Yaskawa INFORM job: slope_planes_program_2.JBI

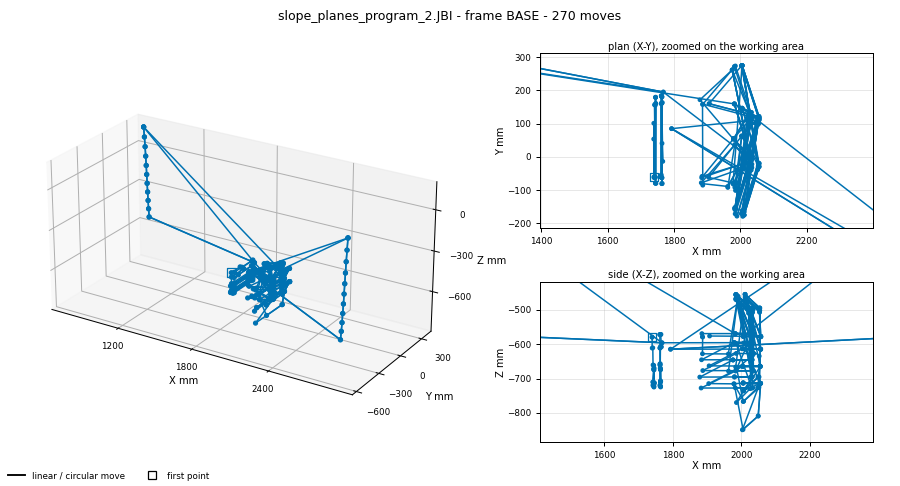
[picture p0: tool path of slope_planes_program_2.JBI in frame BASE, 270 of 278 moves have a stored position in this frame; points joined in program order, loops and branches not executed]
/JOB
//NAME slope_planes_program_2
//POS
///NPOS 270,0,270,0,0,0
///TOOL 0
///POSTYPE BASE
///RECTAN
///RCONF 0,0,0,0,0,0,0,0,0,0,0,0,0,0,0,0,0,0,0,0,0,0,0,0
C00000=1739.260769,-60.871235,-578.989580,5.000000,-89.172678,-175.000000
C00001=1739.028106,53.830840,-579.601277,5.000000,-89.172678,-175.000000
C00002=1739.284791,101.372352,-611.275362,5.000000,-89.172678,-175.000000
C00003=1741.092847,-62.556544,-610.379835,5.000000,-89.172678,-175.000000
C00004=1741.778439,-62.282291,-660.377305,5.000000,-89.172678,-175.000000
C00005=1743.760127,155.636241,-661.504448,5.000000,-89.172678,-175.000000
C00006=1744.673230,178.979946,-711.620985,5.000000,-89.172678,-175.000000
C00007=1740.845557,-59.386621,-710.412050,5.000000,-89.172678,-175.000000
C00008=1743.319095,-61.226324,-673.769949,180.000000,-60.000000,0.000000
C00009=1744.726413,180.007491,-675.029042,180.000000,-60.000000,0.000000
C00010=1744.389872,179.342411,-725.036290,180.000000,-60.000000,0.000000
C00011=1744.215946,-60.947521,-723.764393,180.000000,-60.000000,0.000000
C00012=1884.339610,-58.334513,-568.930098,5.000000,-89.675586,-175.000000
C00013=2032.194970,-12.730020,-568.874909,5.000000,-89.934306,115.240173
C00014=1985.150049,-157.658308,-456.347117,175.000000,-47.917446,5.000000
C00015=2029.012249,-22.244464,-494.713723,175.000000,-65.510944,-60.519673
C00016=2032.887715,-5.143099,-568.885585,5.000000,-89.935736,114.990048
C00017=1981.779671,159.548677,-569.132654,140.189389,-89.999999,5.000000
C00018=2032.201723,-8.373668,-568.883888,-5.000000,-89.934178,115.262595
C00019=1985.641519,-153.780863,-671.511595,-5.000000,-47.740214,-174.961836
C00020=2031.527886,117.688240,-633.513782,5.000000,-65.336014,119.271243
C00021=2033.332423,134.046107,-569.170815,5.000000,-89.932211,115.609393
C00022=1981.779671,159.548677,-569.132654,140.189389,-89.999999,5.000000
C00023=2032.199883,-9.878738,-568.880782,-5.000000,-89.934223,115.254638
C00024=1985.190754,-154.787790,-456.233996,175.000000,-47.916014,5.000000
C00025=2029.085818,-16.497927,-494.609987,175.000000,-65.511330,-60.517922
C00026=2032.946568,0.595729,-568.897051,-5.000000,-89.935689,114.998332
C00027=1981.779671,159.548677,-569.132654,140.189389,-89.999999,5.000000
C00028=2032.202884,-7.055256,-568.886612,5.000000,-89.934137,115.269757
C00029=1985.295997,-151.982336,-466.966556,175.000000,-47.913519,5.000000
C00030=2030.706860,98.840001,-505.585974,175.000000,-65.518281,-60.512478
C00031=2033.557205,115.500512,-569.130752,5.000000,-89.933364,115.405725
C00032=1981.779671,159.548677,-569.132654,140.189389,-89.999999,5.000000
C00033=747.892171,350.982236,154.177497,-16.058325,-5.000000,-175.000000
C00034=747.959774,350.940433,154.234940,-16.059565,-5.000000,-175.000000
C00035=745.781823,361.597631,74.788692,-16.556562,-5.272278,-175.000000
C00036=744.195610,370.293866,-2.453873,-17.385711,-8.680619,-175.000000
C00037=742.808280,377.250152,-77.638846,-18.568266,-11.941707,-175.000000
C00038=742.161890,382.679607,-150.970735,-20.134608,-15.003112,-174.578249
C00039=742.158513,386.664759,-222.101724,-22.108789,-17.810032,-172.917166
C00040=742.703577,389.417825,-291.287358,-24.515478,-20.302282,-171.008190
C00041=744.341698,390.973681,-358.590204,-27.364597,-22.407407,-168.839370
C00042=746.902560,391.345145,-424.326844,-30.640421,-24.064136,-166.421059
C00043=750.369947,390.762543,-488.235309,-34.306804,-25.187057,-163.807677
C00044=755.166090,389.038049,-550.708088,-5.000000,-44.999700,137.718258
C00045=1767.915992,195.255561,-595.676951,140.189389,-89.999999,5.000000
C00046=747.892171,350.982236,154.177497,-16.058325,-5.000000,-175.000000
C00047=747.959774,350.940433,154.234940,-16.059565,-5.000000,-175.000000
C00048=745.781823,361.597631,74.788692,-16.556562,-5.272278,-175.000000
C00049=744.195610,370.293866,-2.453873,-17.385711,-8.680619,-175.000000
C00050=742.808280,377.250152,-77.638846,-18.568266,-11.941707,-175.000000
C00051=742.161890,382.679607,-150.970735,-20.134608,-15.003112,-174.578249
C00052=742.158513,386.664759,-222.101724,-22.108789,-17.810032,-172.917166
C00053=742.703577,389.417825,-291.287358,-24.515478,-20.302282,-171.008190
C00054=744.341698,390.973681,-358.590204,-27.364597,-22.407407,-168.839370
C00055=746.902560,391.345145,-424.326844,-30.640421,-24.064136,-166.421059
C00056=750.369947,390.762543,-488.235309,-34.306804,-25.187057,-163.807677
C00057=755.166090,389.038049,-550.708088,-5.000000,-44.999700,137.718258
C00058=1767.915992,195.255561,-595.676951,140.189389,-89.999999,5.000000
C00059=2030.623854,-5.286374,-595.315431,-5.000000,-89.935275,115.070495
C00060=2026.211755,-22.498761,-494.867644,175.000000,-65.570252,-60.256248
C00061=1983.548198,-157.719294,-455.776356,-175.000000,-47.616753,5.000000
C00062=2030.498190,-12.647404,-595.301228,5.000000,-89.935007,115.117369
C00063=1978.860133,54.290550,-595.350371,140.189389,-89.999999,5.000000
C00064=2030.811257,134.553300,-595.601250,5.000000,-89.935056,115.108749
C00065=2026.562431,117.353936,-508.906406,175.000000,-65.570991,-60.254135
C00066=1983.639451,-153.364957,-469.532259,175.000000,-47.614280,5.000000
C00067=2030.498822,-8.269798,-595.310214,-5.000000,-89.934987,115.120777
C00068=1978.860133,54.290550,-595.350371,140.189389,-89.999999,5.000000
C00069=2030.633524,0.460796,-595.327163,5.000000,-89.935271,115.071236
C00070=2026.217270,-16.752716,-494.764546,-175.000000,-65.570746,-60.254012
C00071=1983.558465,-154.850766,-455.660837,-175.000000,-47.613977,5.000000
C00072=2030.498681,-9.782412,-595.307109,-5.000000,-89.934994,115.119567
C00073=1978.860133,54.290550,-595.350371,140.189389,-89.999999,5.000000
C00074=2030.796749,115.788780,-595.562819,5.000000,-89.935111,115.099123
C00075=2026.507696,98.585677,-505.732438,-175.000000,-65.571101,-60.254277
C00076=1983.625135,-152.033444,-466.398636,175.000000,-47.614083,5.000000
C00077=2030.498875,-6.944594,-595.312935,-5.000000,-89.934981,115.121867
C00078=1978.860133,54.290550,-595.350371,140.189389,-89.999999,5.000000
C00079=1883.381965,-62.373142,-645.345158,5.000000,-89.675586,-175.000000
C00080=2030.706335,-12.453119,-645.300320,5.000000,-89.936548,114.848944
C00081=1983.892004,-157.801574,-454.648135,175.000000,-47.028479,5.000000
C00082=2024.235575,-22.997670,-495.135127,175.000000,-65.680346,-59.751352
C00083=2029.274030,-5.746385,-645.324257,-5.000000,-89.933449,115.390836
C00084=1975.194699,261.761272,-645.797441,140.189389,-89.999999,5.000000
C00085=2030.702768,-8.032373,-645.309265,-5.000000,-89.936754,114.813150
C00086=1983.880333,-153.447358,-468.409969,175.000000,-47.028789,5.000000
C00087=2021.484525,116.857168,-509.189861,-175.000000,-65.680404,-59.751589
C00088=2027.006358,134.400777,-645.623562,5.000000,-89.934799,115.153719
C00089=1975.194699,261.761272,-645.797441,140.189389,-89.999999,5.000000
C00090=2030.703176,-9.560304,-645.306180,-5.000000,-89.936681,114.825864
C00091=1983.830510,-154.932885,-454.540310,175.000000,-47.029501,5.000000
C00092=2024.119139,-17.248911,-495.031310,175.000000,-65.680234,-59.751883
C00093=2029.170564,0.007674,-645.336620,5.000000,-89.933479,115.385431
C00094=1975.194699,261.761272,-645.797441,140.189389,-89.999999,5.000000
C00095=1878.225019,172.061174,-695.855961,5.000000,-89.675586,-175.000000
C00096=2029.216695,-5.923005,-695.325374,5.000000,-89.933075,115.456764
C00097=2023.915349,-23.060021,-495.167917,175.000000,-65.693651,-59.689227
C00098=1983.858125,-157.808143,-454.509625,175.000000,-46.955640,5.000000
C00099=2030.861995,-12.538689,-695.300110,-5.000000,-89.936636,114.833532
C00100=1979.614915,54.878233,-695.349115,140.189389,-89.999999,5.000000
C00101=2026.506483,134.201278,-695.627221,-5.000000,-89.934303,115.240728
C00102=2020.769283,116.793372,-509.225484,175.000000,-65.693966,-59.688064
C00103=1983.837631,-153.454231,-468.268165,175.000000,-46.954194,5.000000
C00104=2030.854062,-8.114311,-695.309074,5.000000,-89.936862,114.794410
C00105=1979.614915,54.878233,-695.349115,140.189389,-89.999999,5.000000
C00106=2029.096697,-0.169123,-695.337832,5.000000,-89.933104,115.451530
C00107=2025.415227,-17.647329,-729.697883,180.000000,-60.000000,0.000000
C00108=1985.252939,-155.837043,-770.197594,180.000000,-60.000000,0.000000
C00109=2030.855920,-9.643522,-695.305982,-5.000000,-89.936782,114.808298
C00110=1979.614915,54.878233,-695.349115,140.189389,-89.999999,5.000000
C00111=1745.307470,160.600706,-712.870295,175.000000,-89.223717,-5.000000
C00112=1745.747004,-79.714542,-714.068825,175.000000,-89.223717,-5.000000
C00113=1743.887926,-78.841577,-670.993376,180.000000,-60.000000,0.000000
C00114=1744.996879,160.942797,-669.818462,180.000000,-60.000000,0.000000
C00115=1741.316004,156.853693,-719.794086,180.000000,-60.000000,0.000000
C00116=1744.102037,-78.968875,-721.002114,180.000000,-60.000000,0.000000
C00117=1885.863395,158.182403,-578.045584,175.000000,-89.336646,-5.000000
C00118=1886.650424,-84.961125,-579.077831,175.000000,-89.336646,-5.000000
C00119=1886.044276,-80.394228,-627.842130,175.000000,-89.336646,-5.000000
C00120=1961.540570,-88.734620,-628.321589,-5.000000,-89.772434,-156.563433
C00121=1989.769528,-39.136527,-460.340640,175.000000,-47.501225,5.075310
C00122=2033.646978,102.591245,-498.881535,175.000000,-65.273893,-60.828128
C00123=2035.991453,119.891152,-627.326416,175.000000,-89.867726,-65.037930
C00124=1984.737237,273.797954,-626.863225,140.054684,-90.000000,5.000000
C00125=1887.028142,158.913088,-676.850323,175.000000,-89.336646,-5.000000
C00126=2034.825328,120.042378,-677.315653,175.000000,-89.867100,-64.984445
C00127=2032.776243,102.409388,-498.967851,175.000000,-65.312424,-60.640081
C00128=1989.800549,-39.182084,-459.925091,175.000000,-47.287692,5.116560
C00129=1962.013642,-91.664127,-678.436686,5.000000,-89.725460,-155.249492
C00130=1982.938067,36.726704,-677.843770,140.054684,-90.000000,5.000000
C00131=2034.622962,-22.049069,-677.911343,175.000000,-89.867279,-64.999786
C00132=2032.449640,-39.666207,-507.153666,-175.000000,-65.312498,-60.640202
C00133=1989.478498,-178.135948,-468.098074,175.000000,-47.287911,5.116557
C00134=2034.502364,-31.953303,-677.951280,175.000000,-89.866766,-64.955929
C00135=1982.938067,36.726704,-677.843770,140.054684,-90.000000,5.000000
C00136=1882.142247,-77.828377,-727.793743,175.000000,-89.336646,-5.000000
C00137=2030.206063,-25.652685,-727.877558,175.000000,-89.864872,-64.793536
C00138=1984.108354,-171.256741,-597.047291,175.000000,-47.594353,5.056180
C00139=2030.104031,98.022525,-634.851776,-175.000000,-65.256846,-60.910378
C00140=2032.751310,115.122397,-727.316773,-175.000000,-89.868050,-65.065618
C00141=1981.628604,272.117578,-726.841892,140.054684,-90.000000,5.000000
C00142=1906.927979,159.938160,-576.005760,175.000000,-88.730027,-5.000000
C00143=2055.823639,120.996000,-576.901902,-175.000000,-89.740938,-65.240948
C00144=2053.106317,103.764595,-494.268027,-175.000000,-65.230923,-61.019642
C00145=2010.474853,-34.355523,-454.220693,175.000000,-46.647438,5.000000
C00146=2056.406479,111.482410,-576.995998,175.000000,-89.745867,-65.461252
C00147=2005.209070,146.661390,-577.065002,139.450504,-90.000000,5.000000
C00148=2055.842019,116.746081,-576.937074,-175.000000,-89.740871,-65.237935
C00149=2052.989906,99.574050,-500.952961,175.000000,-65.230260,-61.021788
C00150=2011.168552,-174.704832,-462.043828,175.000000,-46.649165,5.000000
C00151=2056.691524,-29.178943,-578.150938,175.000000,-89.740607,-65.226111
C00152=2005.209070,146.661390,-577.065002,139.450504,-90.000000,5.000000
C00153=2055.849079,115.132278,-576.950432,175.000000,-89.740846,-65.236825
C00154=2052.885022,98.006554,-506.182198,175.000000,-65.231218,-61.022508
C00155=2010.996515,-165.146838,-467.177110,175.000000,-46.648598,5.000000
C00156=2056.648001,-19.660442,-578.072096,-175.000000,-89.740735,-65.231870
C00157=2005.209070,146.661390,-577.065002,139.450504,-90.000000,5.000000
C00158=2926.142829,-568.766451,147.287214,16.077910,5.000000,-175.000000
C00159=2926.076134,-568.725021,147.346073,16.079159,5.000000,-175.000000
C00160=2926.915259,-579.012665,67.975421,16.618272,5.069146,-175.000000
C00161=2927.180823,-587.344273,-9.172130,17.488477,8.466523,-175.000000
C00162=2927.263613,-593.939517,-84.251280,18.710876,11.711988,-175.000000
C00163=2926.618715,-599.009172,-157.460463,20.315045,14.752889,-174.614405
C00164=2925.350749,-602.637128,-228.455516,22.323798,17.534410,-172.947796
C00165=2923.550953,-605.033416,-297.496048,24.760039,19.996597,-171.037121
C00166=2920.674981,-606.231856,-364.637283,27.631362,22.067786,-168.873373
C00167=2916.889432,-606.243200,-430.199558,30.919773,23.688222,-166.469791
C00168=2912.216145,-605.298605,-493.924262,34.586747,24.774919,-163.883699
C00169=2906.228082,-603.207784,-556.196538,5.000000,-44.999700,-43.020627
C00170=1792.874536,85.158203,-614.480492,139.450504,-90.000000,5.000000
C00171=2926.142829,-568.766451,147.287214,16.077910,5.000000,-175.000000
C00172=2926.076134,-568.725021,147.346073,16.079159,5.000000,-175.000000
C00173=2926.915259,-579.012665,67.975421,16.618272,5.069146,-175.000000
C00174=2927.180823,-587.344273,-9.172130,17.488477,8.466523,-175.000000
C00175=2927.263613,-593.939517,-84.251280,18.710876,11.711988,-175.000000
C00176=2926.618715,-599.009172,-157.460463,20.315045,14.752889,-174.614405
C00177=2925.350749,-602.637128,-228.455516,22.323798,17.534410,-172.947796
C00178=2923.550953,-605.033416,-297.496048,24.760039,19.996597,-171.037121
C00179=2920.674981,-606.231856,-364.637283,27.631362,22.067786,-168.873373
C00180=2916.889432,-606.243200,-430.199558,30.919773,23.688222,-166.469791
C00181=2912.216145,-605.298605,-493.924262,34.586747,24.774919,-163.883699
C00182=2906.228082,-603.207784,-556.196538,5.000000,-44.999700,-43.020627
C00183=1792.874536,85.158203,-614.480492,139.450504,-90.000000,5.000000
C00184=2056.365022,112.180676,-614.060084,175.000000,-89.754111,-65.826891
C00185=2010.304299,-34.348003,-454.300976,-175.000000,-46.690667,5.000000
C00186=2053.113251,103.801510,-494.249331,175.000000,-65.223766,-61.057680
C00187=2054.950475,121.310524,-613.945356,-175.000000,-89.741164,-65.251079
C00188=2003.613875,274.609972,-613.046909,139.450504,-90.000000,5.000000
C00189=2055.636711,-28.833132,-615.190528,175.000000,-89.741469,-65.264777
C00190=2010.762539,-174.697243,-462.120527,175.000000,-46.693233,5.000000
C00191=2052.989855,99.611187,-500.934525,175.000000,-65.223279,-61.059877
C00192=2054.963740,117.061501,-613.980420,-175.000000,-89.741115,-65.248883
C00193=2003.613875,274.609972,-613.046909,139.450504,-90.000000,5.000000
C00194=2055.611620,-19.313431,-615.112101,175.000000,-89.741623,-65.271640
C00195=2010.606196,-165.141325,-467.254668,175.000000,-46.692932,5.000000
C00196=2052.880597,98.042038,-506.162006,-175.000000,-65.223525,-61.059754
C00197=2054.968836,115.448028,-613.993736,175.000000,-89.741097,-65.248074
C00198=2003.613875,274.609972,-613.046909,139.450504,-90.000000,5.000000
C00199=1905.444423,160.394797,-663.048331,175.000000,-88.730027,-5.000000
C00200=2054.288678,121.721853,-663.941303,175.000000,-89.741203,-65.252828
C00201=2053.572048,103.808577,-494.255875,175.000000,-65.222389,-61.064975
C00202=2010.729321,-34.346497,-454.326314,175.000000,-46.698848,5.000000
C00203=1982.997461,-91.393846,-666.556684,5.000000,-89.290634,-153.408707
C00204=2003.833524,62.704577,-664.801360,139.450504,-90.000000,5.000000
C00205=2054.301207,117.472936,-663.976351,175.000000,-89.741156,-65.250728
C00206=2053.441415,99.615968,-500.942181,175.000000,-65.222387,-61.064778
C00207=2011.161552,-174.696248,-462.139956,-175.000000,-46.698673,5.000000
C00208=2055.017240,-28.386626,-665.187598,-175.000000,-89.742226,-65.298653
C00209=2003.833524,62.704577,-664.801360,139.450504,-90.000000,5.000000
C00210=2054.298510,118.381369,-663.968857,175.000000,-89.741166,-65.251169
C00211=2047.226085,101.805884,-726.798896,180.000000,-60.000000,0.000000
C00212=2005.084758,-36.143454,-767.317247,180.000000,-60.000000,0.000000
C00213=1985.146296,-100.782685,-667.019520,5.000000,-89.130627,-151.651480
C00214=2003.833524,62.704577,-664.801360,139.450504,-90.000000,5.000000
C00215=2054.306022,115.859502,-663.989661,175.000000,-89.741139,-65.249954
C00216=2047.942670,99.027002,-695.065787,180.000000,-60.000000,0.000000
C00217=2006.305061,-161.985001,-736.601336,180.000000,-60.000000,0.000000
C00218=2055.004793,-18.862115,-665.109477,175.000000,-89.742478,-65.309922
C00219=2003.833524,62.704577,-664.801360,139.450504,-90.000000,5.000000
C00220=1904.312540,-61.480856,-714.854482,175.000000,-88.730027,-5.000000
C00221=1978.599133,-78.361413,-715.611563,5.000000,-89.666032,-158.688293
C00222=2004.663042,-30.081199,-848.850205,180.000000,-60.000000,0.000000
C00223=2048.840642,106.231449,-809.568616,180.000000,-60.000000,0.000000
C00224=2055.976206,122.261173,-713.990008,175.000000,-89.743857,-65.371606
C00225=2005.159554,275.098461,-713.105097,139.450504,-90.000000,5.000000
C00226=2053.250187,-28.118095,-715.158302,-175.000000,-89.739361,-65.170219
C00227=2002.563508,-170.486237,-849.835390,180.000000,-60.000000,0.000000
C00228=2048.782161,101.984317,-809.485547,180.000000,-60.000000,0.000000
C00229=2055.929750,118.022396,-714.023803,-175.000000,-89.744018,-65.378790
C00230=2005.159554,275.098461,-713.105097,139.450504,-90.000000,5.000000
C00231=1977.602007,-81.260640,-715.503831,5.000000,-89.723124,-159.673738
C00232=2006.414048,-36.066539,-766.392101,180.000000,-60.000000,0.000000
C00233=2050.619682,102.216611,-727.093987,180.000000,-60.000000,0.000000
C00234=2055.939745,118.928698,-714.016579,175.000000,-89.743984,-65.377280
C00235=2005.159554,275.098461,-713.105097,139.450504,-90.000000,5.000000
C00236=2053.225132,-33.321148,-715.200690,175.000000,-89.739860,-65.192600
C00237=2006.882768,-178.738220,-595.871797,175.000000,-47.198218,5.000000
C00238=2051.802734,-38.380071,-634.637018,175.000000,-65.138912,-61.504047
C00239=2054.163138,-21.335497,-715.128058,175.000000,-89.747043,-65.513648
C00240=2005.159554,275.098461,-713.105097,139.450504,-90.000000,5.000000
C00241=2053.282810,-18.656752,-715.080857,175.000000,-89.738334,-65.124025
C00242=2005.240768,-161.906151,-735.627370,180.000000,-60.000000,0.000000
C00243=2051.290198,99.439970,-695.357513,180.000000,-60.000000,0.000000
C00244=2055.911917,116.412698,-714.036631,175.000000,-89.744078,-65.381437
C00245=2005.159554,275.098461,-713.105097,139.450504,-90.000000,5.000000
C00246=1764.879905,163.737879,-571.172420,-175.000000,-89.333764,-5.000000
C00247=1764.057547,40.943257,-571.686752,-175.000000,-89.333764,-5.000000
C00248=1766.307154,-13.323645,-607.577811,-175.000000,-89.333764,-5.000000
C00249=1763.380971,162.239603,-606.794756,-175.000000,-89.333764,-5.000000
C00250=1762.810953,161.810268,-656.793795,-175.000000,-89.333764,-5.000000
C00251=1761.795682,-53.749228,-657.701658,-175.000000,-89.333764,-5.000000
C00252=1764.265859,-79.604216,-707.844526,-175.000000,-89.333764,-5.000000
C00253=1763.258444,162.029582,-706.801898,-175.000000,-89.333764,-5.000000
C00254=1762.681818,161.610046,-670.198278,180.000000,-60.000000,0.000000
C00255=1763.869591,-80.392370,-671.244576,180.000000,-60.000000,0.000000
C00256=1763.310066,-80.290661,-721.241471,180.000000,-60.000000,0.000000
C00257=1761.532878,159.749711,-720.196690,180.000000,-60.000000,0.000000
C00258=1761.566018,-60.389450,-571.247562,5.000000,-89.445806,-175.000000
C00259=1761.583926,184.103056,-572.110136,5.000000,-89.445806,-175.000000
C00260=1762.248770,183.727510,-611.406244,5.000000,-89.445806,-175.000000
C00261=1761.627598,-60.731547,-610.549624,5.000000,-89.445806,-175.000000
C00262=1762.073443,-61.075018,-660.546750,5.000000,-89.445806,-175.000000
C00263=1762.413537,182.923131,-661.404463,5.000000,-89.445806,-175.000000
C00264=1763.161347,182.417921,-711.398097,5.000000,-89.445806,-175.000000
C00265=1763.254633,-62.409155,-710.533267,5.000000,-89.445806,-175.000000
C00266=1763.389680,-62.871249,-673.930440,180.000000,-60.000000,0.000000
C00267=1763.610457,181.502527,-674.790632,180.000000,-60.000000,0.000000
C00268=1763.838836,180.206390,-724.786500,180.000000,-60.000000,0.000000
C00269=1763.938440,-62.435048,-723.929321,180.000000,-60.000000,0.000000
///POSTYPE PULSE
///PULSE
EC00000=51200.0
EC00001=51200.0
EC00002=51200.0
EC00003=51200.0
EC00004=51200.0
EC00005=51200.0
EC00006=51200.0
EC00007=51200.0
EC00008=51200.0
EC00009=51200.0
EC00010=51200.0
EC00011=51200.0
EC00012=51200.0
EC00013=51200.0
EC00014=51200.0
EC00015=51200.0
EC00016=51200.0
EC00017=51200.0
EC00018=51200.0
EC00019=51200.0
EC00020=51200.0
EC00021=51200.0
EC00022=51200.0
EC00023=51200.0
EC00024=51200.0
EC00025=51200.0
EC00026=51200.0
EC00027=51200.0
EC00028=51200.0
EC00029=51200.0
EC00030=51200.0
EC00031=51200.0
EC00032=51200.0
EC00033=51200.0
EC00034=51200.0
EC00035=51200.0
EC00036=51200.0
EC00037=51200.0
EC00038=51200.0
EC00039=51200.0
EC00040=51200.0
EC00041=51200.0
EC00042=51200.0
EC00043=51200.0
EC00044=51200.0
EC00045=51200.0
EC00046=51200.0
EC00047=51200.0
EC00048=51200.0
EC00049=51200.0
EC00050=51200.0
EC00051=51200.0
EC00052=51200.0
EC00053=51200.0
EC00054=51200.0
EC00055=51200.0
EC00056=51200.0
EC00057=51200.0
EC00058=51200.0
EC00059=51200.0
EC00060=51200.0
EC00061=51200.0
EC00062=51200.0
EC00063=51200.0
EC00064=51200.0
EC00065=51200.0
EC00066=51200.0
EC00067=51200.0
EC00068=51200.0
EC00069=51200.0
EC00070=51200.0
EC00071=51200.0
EC00072=51200.0
EC00073=51200.0
EC00074=51200.0
EC00075=51200.0
EC00076=51200.0
EC00077=51200.0
EC00078=51200.0
EC00079=51200.0
EC00080=51200.0
EC00081=51200.0
EC00082=51200.0
EC00083=51200.0
EC00084=51200.0
EC00085=51200.0
EC00086=51200.0
EC00087=51200.0
EC00088=51200.0
EC00089=51200.0
EC00090=51200.0
EC00091=51200.0
EC00092=51200.0
EC00093=51200.0
EC00094=51200.0
EC00095=51200.0
EC00096=51200.0
EC00097=51200.0
EC00098=51200.0
EC00099=51200.0
EC00100=51200.0
EC00101=51200.0
EC00102=51200.0
EC00103=51200.0
EC00104=51200.0
EC00105=51200.0
EC00106=51200.0
EC00107=51200.0
EC00108=51200.0
EC00109=51200.0
EC00110=51200.0
EC00111=143360.0
EC00112=143360.0
EC00113=143360.0
EC00114=143360.0
EC00115=143360.0
EC00116=143360.0
EC00117=143360.0
EC00118=143360.0
EC00119=143360.0
EC00120=143360.0
EC00121=143360.0
EC00122=143360.0
EC00123=143360.0
EC00124=143360.0
EC00125=143360.0
EC00126=143360.0
EC00127=143360.0
EC00128=143360.0
EC00129=143360.0
EC00130=143360.0
EC00131=143360.0
EC00132=143360.0
EC00133=143360.0
EC00134=143360.0
EC00135=143360.0
EC00136=143360.0
EC00137=143360.0
EC00138=143360.0
EC00139=143360.0
EC00140=143360.0
EC00141=143360.0
EC00142=234496.0
EC00143=234496.0
EC00144=234496.0
EC00145=234496.0
EC00146=234496.0
EC00147=234496.0
EC00148=234496.0
EC00149=234496.0
EC00150=234496.0
EC00151=234496.0
EC00152=234496.0
EC00153=234496.0
EC00154=234496.0
EC00155=234496.0
EC00156=234496.0
EC00157=234496.0
EC00158=234496.0
EC00159=234496.0
EC00160=234496.0
EC00161=234496.0
EC00162=234496.0
EC00163=234496.0
EC00164=234496.0
EC00165=234496.0
EC00166=234496.0
EC00167=234496.0
EC00168=234496.0
EC00169=234496.0
EC00170=234496.0
EC00171=234496.0
EC00172=234496.0
EC00173=234496.0
EC00174=234496.0
EC00175=234496.0
EC00176=234496.0
EC00177=234496.0
EC00178=234496.0
EC00179=234496.0
EC00180=234496.0
EC00181=234496.0
EC00182=234496.0
EC00183=234496.0
EC00184=234496.0
EC00185=234496.0
EC00186=234496.0
EC00187=234496.0
EC00188=234496.0
EC00189=234496.0
EC00190=234496.0
EC00191=234496.0
EC00192=234496.0
EC00193=234496.0
EC00194=234496.0
EC00195=234496.0
EC00196=234496.0
EC00197=234496.0
EC00198=234496.0
EC00199=234496.0
EC00200=234496.0
EC00201=234496.0
EC00202=234496.0
EC00203=234496.0
EC00204=234496.0
EC00205=234496.0
EC00206=234496.0
EC00207=234496.0
EC00208=234496.0
EC00209=234496.0
EC00210=234496.0
EC00211=234496.0
EC00212=234496.0
EC00213=234496.0
EC00214=234496.0
EC00215=234496.0
EC00216=234496.0
EC00217=234496.0
EC00218=234496.0
EC00219=234496.0
EC00220=234496.0
EC00221=234496.0
EC00222=234496.0
EC00223=234496.0
EC00224=234496.0
EC00225=234496.0
EC00226=234496.0
EC00227=234496.0
EC00228=234496.0
EC00229=234496.0
EC00230=234496.0
EC00231=234496.0
EC00232=234496.0
EC00233=234496.0
EC00234=234496.0
EC00235=234496.0
EC00236=234496.0
EC00237=234496.0
EC00238=234496.0
EC00239=234496.0
EC00240=234496.0
EC00241=234496.0
EC00242=234496.0
EC00243=234496.0
EC00244=234496.0
EC00245=234496.0
EC00246=235520.0
EC00247=235520.0
EC00248=235520.0
EC00249=235520.0
EC00250=235520.0
EC00251=235520.0
EC00252=235520.0
EC00253=235520.0
EC00254=235520.0
EC00255=235520.0
EC00256=235520.0
EC00257=235520.0
EC00258=327680.0
EC00259=327680.0
EC00260=327680.0
EC00261=327680.0
EC00262=327680.0
EC00263=327680.0
EC00264=327680.0
EC00265=327680.0
EC00266=327680.0
EC00267=327680.0
EC00268=327680.0
EC00269=327680.0
//INST
///DATE 2023/08/13 11:59
///ATTR SC,RW,RJ
////FRAME BASE
///GROUP1 RB1,ST1
NOP
MOVJ P009 EX000 VJ=15.00
MOVJ C00000 EC00000 VJ=15.0
CALL JOB:SPYON
MOVL C00001 EC00001 V=150.0
MOVL C00002 EC00002 V=150.0
MOVL C00003 EC00003 V=150.0
MOVL C00004 EC00004 V=150.0
MOVL C00005 EC00005 V=150.0
MOVL C00006 EC00006 V=150.0
MOVL C00007 EC00007 V=150.0
MOVL C00008 EC00008 V=150.0
MOVL C00009 EC00009 V=150.0
MOVL C00010 EC00010 V=150.0
MOVL C00011 EC00011 V=150.0
CALL JOB:SPYOF
MOVJ P009 VJ=15.00
MOVJ C00012 EC00012 VJ=15.0
CALL JOB:SPYON
MOVL C00013 EC00013 V=150.0
MOVL C00014 EC00014 V=150.0
MOVL C00015 EC00015 V=150.0
MOVL C00016 EC00016 V=150.0
MOVL C00017 EC00017 V=150.0
MOVL C00018 EC00018 V=150.0
MOVL C00019 EC00019 V=150.0
MOVL C00020 EC00020 V=150.0
MOVL C00021 EC00021 V=150.0
MOVL C00022 EC00022 V=150.0
MOVL C00023 EC00023 V=150.0
MOVL C00024 EC00024 V=150.0
MOVL C00025 EC00025 V=150.0
MOVL C00026 EC00026 V=150.0
MOVL C00027 EC00027 V=150.0
MOVL C00028 EC00028 V=150.0
MOVL C00029 EC00029 V=150.0
MOVL C00030 EC00030 V=150.0
MOVL C00031 EC00031 V=150.0
MOVL C00032 EC00032 V=150.0
MOVL C00033 EC00033 V=150.0
MOVL C00034 EC00034 V=150.0
MOVL C00035 EC00035 V=150.0
MOVL C00036 EC00036 V=150.0
MOVL C00037 EC00037 V=150.0
MOVL C00038 EC00038 V=150.0
MOVL C00039 EC00039 V=150.0
MOVL C00040 EC00040 V=150.0
MOVL C00041 EC00041 V=150.0
MOVL C00042 EC00042 V=150.0
MOVL C00043 EC00043 V=150.0
MOVL C00044 EC00044 V=150.0
MOVL C00045 EC00045 V=150.0
MOVL C00046 EC00046 V=150.0
MOVL C00047 EC00047 V=150.0
MOVL C00048 EC00048 V=150.0
MOVL C00049 EC00049 V=150.0
MOVL C00050 EC00050 V=150.0
MOVL C00051 EC00051 V=150.0
MOVL C00052 EC00052 V=150.0
MOVL C00053 EC00053 V=150.0
MOVL C00054 EC00054 V=150.0
MOVL C00055 EC00055 V=150.0
MOVL C00056 EC00056 V=150.0
MOVL C00057 EC00057 V=150.0
MOVL C00058 EC00058 V=150.0
MOVL C00059 EC00059 V=150.0
MOVL C00060 EC00060 V=150.0
MOVL C00061 EC00061 V=150.0
MOVL C00062 EC00062 V=150.0
MOVL C00063 EC00063 V=150.0
MOVL C00064 EC00064 V=150.0
MOVL C00065 EC00065 V=150.0
MOVL C00066 EC00066 V=150.0
MOVL C00067 EC00067 V=150.0
MOVL C00068 EC00068 V=150.0
MOVL C00069 EC00069 V=150.0
MOVL C00070 EC00070 V=150.0
MOVL C00071 EC00071 V=150.0
MOVL C00072 EC00072 V=150.0
MOVL C00073 EC00073 V=150.0
MOVL C00074 EC00074 V=150.0
MOVL C00075 EC00075 V=150.0
MOVL C00076 EC00076 V=150.0
MOVL C00077 EC00077 V=150.0
MOVL C00078 EC00078 V=150.0
MOVL C00079 EC00079 V=150.0
MOVL C00080 EC00080 V=150.0
MOVL C00081 EC00081 V=150.0
MOVL C00082 EC00082 V=150.0
MOVL C00083 EC00083 V=150.0
MOVL C00084 EC00084 V=150.0
MOVL C00085 EC00085 V=150.0
MOVL C00086 EC00086 V=150.0
MOVL C00087 EC00087 V=150.0
MOVL C00088 EC00088 V=150.0
MOVL C00089 EC00089 V=150.0
MOVL C00090 EC00090 V=150.0
MOVL C00091 EC00091 V=150.0
MOVL C00092 EC00092 V=150.0
MOVL C00093 EC00093 V=150.0
MOVL C00094 EC00094 V=150.0
MOVL C00095 EC00095 V=150.0
MOVL C00096 EC00096 V=150.0
MOVL C00097 EC00097 V=150.0
MOVL C00098 EC00098 V=150.0
MOVL C00099 EC00099 V=150.0
MOVL C00100 EC00100 V=150.0
MOVL C00101 EC00101 V=150.0
MOVL C00102 EC00102 V=150.0
MOVL C00103 EC00103 V=150.0
MOVL C00104 EC00104 V=150.0
MOVL C00105 EC00105 V=150.0
MOVL C00106 EC00106 V=150.0
MOVL C00107 EC00107 V=150.0
MOVL C00108 EC00108 V=150.0
MOVL C00109 EC00109 V=150.0
MOVL C00110 EC00110 V=150.0
CALL JOB:SPYOF
MOVJ P009 VJ=15.00
MOVJ C00111 EC00111 VJ=15.0
CALL JOB:SPYON
MOVL C00112 EC00112 V=150.0
MOVL C00113 EC00113 V=150.0
MOVL C00114 EC00114 V=150.0
MOVL C00115 EC00115 V=150.0
MOVL C00116 EC00116 V=150.0
CALL JOB:SPYOF
MOVJ P009 VJ=15.00
MOVJ C00117 EC00117 VJ=15.0
CALL JOB:SPYON
MOVL C00118 EC00118 V=150.0
MOVL C00119 EC00119 V=150.0
MOVL C00120 EC00120 V=150.0
MOVL C00121 EC00121 V=150.0
MOVL C00122 EC00122 V=150.0
MOVL C00123 EC00123 V=150.0
MOVL C00124 EC00124 V=150.0
MOVL C00125 EC00125 V=150.0
MOVL C00126 EC00126 V=150.0
MOVL C00127 EC00127 V=150.0
MOVL C00128 EC00128 V=150.0
MOVL C00129 EC00129 V=150.0
MOVL C00130 EC00130 V=150.0
MOVL C00131 EC00131 V=150.0
MOVL C00132 EC00132 V=150.0
MOVL C00133 EC00133 V=150.0
MOVL C00134 EC00134 V=150.0
MOVL C00135 EC00135 V=150.0
MOVL C00136 EC00136 V=150.0
MOVL C00137 EC00137 V=150.0
MOVL C00138 EC00138 V=150.0
MOVL C00139 EC00139 V=150.0
MOVL C00140 EC00140 V=150.0
MOVL C00141 EC00141 V=150.0
CALL JOB:SPYOF
MOVJ P009 VJ=15.00
MOVJ C00142 EC00142 VJ=15.0
CALL JOB:SPYON
MOVL C00143 EC00143 V=150.0
MOVL C00144 EC00144 V=150.0
MOVL C00145 EC00145 V=150.0
MOVL C00146 EC00146 V=150.0
MOVL C00147 EC00147 V=150.0
MOVL C00148 EC00148 V=150.0
MOVL C00149 EC00149 V=150.0
MOVL C00150 EC00150 V=150.0
MOVL C00151 EC00151 V=150.0
MOVL C00152 EC00152 V=150.0
MOVL C00153 EC00153 V=150.0
MOVL C00154 EC00154 V=150.0
MOVL C00155 EC00155 V=150.0
MOVL C00156 EC00156 V=150.0
MOVL C00157 EC00157 V=150.0
MOVL C00158 EC00158 V=150.0
MOVL C00159 EC00159 V=150.0
MOVL C00160 EC00160 V=150.0
MOVL C00161 EC00161 V=150.0
MOVL C00162 EC00162 V=150.0
MOVL C00163 EC00163 V=150.0
MOVL C00164 EC00164 V=150.0
MOVL C00165 EC00165 V=150.0
MOVL C00166 EC00166 V=150.0
MOVL C00167 EC00167 V=150.0
MOVL C00168 EC00168 V=150.0
MOVL C00169 EC00169 V=150.0
MOVL C00170 EC00170 V=150.0
MOVL C00171 EC00171 V=150.0
MOVL C00172 EC00172 V=150.0
MOVL C00173 EC00173 V=150.0
MOVL C00174 EC00174 V=150.0
MOVL C00175 EC00175 V=150.0
MOVL C00176 EC00176 V=150.0
MOVL C00177 EC00177 V=150.0
MOVL C00178 EC00178 V=150.0
MOVL C00179 EC00179 V=150.0
MOVL C00180 EC00180 V=150.0
MOVL C00181 EC00181 V=150.0
MOVL C00182 EC00182 V=150.0
MOVL C00183 EC00183 V=150.0
MOVL C00184 EC00184 V=150.0
MOVL C00185 EC00185 V=150.0
MOVL C00186 EC00186 V=150.0
MOVL C00187 EC00187 V=150.0
MOVL C00188 EC00188 V=150.0
MOVL C00189 EC00189 V=150.0
MOVL C00190 EC00190 V=150.0
MOVL C00191 EC00191 V=150.0
MOVL C00192 EC00192 V=150.0
MOVL C00193 EC00193 V=150.0
MOVL C00194 EC00194 V=150.0
MOVL C00195 EC00195 V=150.0
MOVL C00196 EC00196 V=150.0
MOVL C00197 EC00197 V=150.0
MOVL C00198 EC00198 V=150.0
MOVL C00199 EC00199 V=150.0
MOVL C00200 EC00200 V=150.0
MOVL C00201 EC00201 V=150.0
MOVL C00202 EC00202 V=150.0
MOVL C00203 EC00203 V=150.0
MOVL C00204 EC00204 V=150.0
MOVL C00205 EC00205 V=150.0
MOVL C00206 EC00206 V=150.0
MOVL C00207 EC00207 V=150.0
MOVL C00208 EC00208 V=150.0
MOVL C00209 EC00209 V=150.0
MOVL C00210 EC00210 V=150.0
MOVL C00211 EC00211 V=150.0
MOVL C00212 EC00212 V=150.0
MOVL C00213 EC00213 V=150.0
MOVL C00214 EC00214 V=150.0
MOVL C00215 EC00215 V=150.0
MOVL C00216 EC00216 V=150.0
MOVL C00217 EC00217 V=150.0
MOVL C00218 EC00218 V=150.0
MOVL C00219 EC00219 V=150.0
MOVL C00220 EC00220 V=150.0
MOVL C00221 EC00221 V=150.0
MOVL C00222 EC00222 V=150.0
MOVL C00223 EC00223 V=150.0
MOVL C00224 EC00224 V=150.0
MOVL C00225 EC00225 V=150.0
MOVL C00226 EC00226 V=150.0
MOVL C00227 EC00227 V=150.0
MOVL C00228 EC00228 V=150.0
MOVL C00229 EC00229 V=150.0
MOVL C00230 EC00230 V=150.0
MOVL C00231 EC00231 V=150.0
MOVL C00232 EC00232 V=150.0
MOVL C00233 EC00233 V=150.0
MOVL C00234 EC00234 V=150.0
MOVL C00235 EC00235 V=150.0
MOVL C00236 EC00236 V=150.0
MOVL C00237 EC00237 V=150.0
MOVL C00238 EC00238 V=150.0
MOVL C00239 EC00239 V=150.0
MOVL C00240 EC00240 V=150.0
MOVL C00241 EC00241 V=150.0
MOVL C00242 EC00242 V=150.0
MOVL C00243 EC00243 V=150.0
MOVL C00244 EC00244 V=150.0
MOVL C00245 EC00245 V=150.0
CALL JOB:SPYOF
MOVJ P009 VJ=15.00
MOVJ C00246 EC00246 VJ=15.0
CALL JOB:SPYON
MOVL C00247 EC00247 V=150.0
MOVL C00248 EC00248 V=150.0
MOVL C00249 EC00249 V=150.0
MOVL C00250 EC00250 V=150.0
MOVL C00251 EC00251 V=150.0
MOVL C00252 EC00252 V=150.0
MOVL C00253 EC00253 V=150.0
MOVL C00254 EC00254 V=150.0
MOVL C00255 EC00255 V=150.0
MOVL C00256 EC00256 V=150.0
MOVL C00257 EC00257 V=150.0
CALL JOB:SPYOF
MOVJ P009 VJ=15.00
MOVJ C00258 EC00258 VJ=15.0
CALL JOB:SPYON
MOVL C00259 EC00259 V=150.0
MOVL C00260 EC00260 V=150.0
MOVL C00261 EC00261 V=150.0
MOVL C00262 EC00262 V=150.0
MOVL C00263 EC00263 V=150.0
MOVL C00264 EC00264 V=150.0
MOVL C00265 EC00265 V=150.0
MOVL C00266 EC00266 V=150.0
MOVL C00267 EC00267 V=150.0
MOVL C00268 EC00268 V=150.0
MOVL C00269 EC00269 V=150.0
CALL JOB:SPYOF
MOVJ P009 VJ=15.00
END
